FUNCTION_BLOCK FB_Visualization
VAR_INPUT
	bMovingRight : BOOL;
	bMovingLeft : BOOL;
END_VAR
VAR_OUTPUT
	bLimitLeft : BOOL;
	bLimitRight: BOOL;
END_VAR
VAR
	Position: REAL;
END_VAR

IF bMovingRight THEN
	bLimitLeft := FALSE;
	bLimitRight := FALSE;
	Position := Position + 0.5;
	IF (Position >= 310) THEN
		bLimitRight := TRUE;
	END_IF
ELSIF bMovingLeft THEN
	bLimitLeft := FALSE;
	bLimitRight := FALSE;
	Position := Position - 0.5;
	IF (Position <=  0) THEN
		bLimitLeft := TRUE;
	END_IF
END_IF

END_FUNCTION_BLOCK

(* stored: Version 1.1.0.1, ProductVersion 3.1.4024.12
   POU FB_Visualization: Id {ea6cfb47-13fc-4b28-af4c-16077307fb77}, SpecialFunc None *)
